PROGRAM MOVE_TO_POSITION
VAR CONSTANT
	UP_OFFSET : REAL :=-1.375;
	DOWN_OFFSET : REAL := 0.675;
	POSITION_SCALE : REAL := 12000;
END_VAR
VAR
	currentRawPosition AT %I* : UDINT;
	
END_VAR

GV_LIFT.CURRENT_POSITION := UDINT_TO_REAL(currentRawPosition) / POSITION_SCALE;

IF (GV_LIFT.RUN_BUTTON_OUT) AND GV_LIFT.MTS_ALLOWED	THEN
	IF(GV_LIFT.CURRENT_POSITION > (GV_LIFT.TARGET_POSITION + DOWN_OFFSET)) THEN
		GV_LIFT.DOWN_BUTTON_OUT := TRUE;
		GV_LIFT.JUST_RAN := TRUE;
	ELSIF(GV_LIFT.CURRENT_POSITION < (GV_LIFT.TARGET_POSITION + UP_OFFSET)) THEN
		GV_LIFT.UP_BUTTON_OUT := TRUE;
		GV_LIFT.JUST_RAN := TRUE;
	ELSE
		GV_LIFT.UP_BUTTON_OUT := FALSE;
		GV_LIFT.DOWN_BUTTON_OUT := FALSE;
		GV_LIFT.MTS_ALLOWED := FALSE;
		GV_LIFT.JUST_RAN:= FALSE;
	END_IF
ELSIF GV_LIFT.JUST_RAN THEN
		GV_LIFT.MTS_ALLOWED := FALSE;
	
END_IF

END_PROGRAM

(* stored: Version 1.1.0.1, ProductVersion 3.1.4022.12
   POU MOVE_TO_POSITION: Id {56c13076-a9dd-4c45-b27c-b090b1590a60}, SpecialFunc None *)
